{attribute 'linkalways'} 
{attribute 'no_explicit_call' := 'This FB is a CLASS and must be accessed using methods or properties'}
{attribute 'enable_dynamic_creation'}
FUNCTION_BLOCK GetBlueprintVisitor EXTENDS Disposable IMPLEMENTS I_NodePrototypeVisitor
VAR
	serializer : JsonSerializer;
END_VAR

METHOD VisitContent
VAR_INPUT
	VisitingContent : I_Content;
END_VAR
END_METHOD

METHOD VisitError
VAR_INPUT
	VisitingError : I_Alarm;
END_VAR
END_METHOD

METHOD VisitExtension
VAR_INPUT
	VisitingExtension : I_Extension;
END_VAR
END_METHOD

METHOD VisitInputPort
VAR_INPUT
	VisitingInputPort : I_InputPort;
END_VAR
END_METHOD

METHOD VisitMetadatum
VAR_INPUT
	VisitingMetadatum : I_Metadata;
END_VAR
END_METHOD

METHOD VisitNode
VAR_INPUT
	VisitingNode : I_Node;
END_VAR
serializer.StartObject();
END_METHOD

METHOD VisitOutputPort
VAR_INPUT
	VisitingOutputPort : I_OutputPort;
END_VAR
END_METHOD

METHOD VisitParameter
VAR_INPUT
	VisitingProperty : I_Parameter;
END_VAR
END_METHOD

METHOD VisitPrototype
VAR_INPUT
	VisitingPrototype : I_NodePrototype;
END_VAR
serializer.Reset();
serializer.StartObject();
serializer.AddKey('blueprints');
serializer.StartArray();

serializer.EndArray();
serializer.EndObject();
END_METHOD

END_FUNCTION_BLOCK

(* stored: Version 1.1.0.1, ProductVersion 3.1.4024.12
   POU GetBlueprintVisitor: Id {9f9a0116-9d81-4a08-a879-7a2851d51385}, SpecialFunc None
   Method VisitContent: Id {5d6b8e87-493f-4bc0-a416-bdda199c430d}
   Method VisitError: Id {08d6423b-3444-4d02-ae95-4e4c7fed218c}
   Method VisitExtension: Id {4b74c9d7-8e37-404e-add7-587af0696243}
   Method VisitInputPort: Id {0763b377-826e-4b34-9135-9701e00da90a}
   Method VisitMetadatum: Id {69ef5793-7e33-4a4a-bd31-0b8a852dd40c}
   Method VisitNode: Id {0c574603-4091-4b53-bc43-a99c409aff80}
   Method VisitOutputPort: Id {08afcd2c-2b3e-40a2-8371-470084bdd009}
   Method VisitParameter: Id {cb761164-ab6e-4c1f-a1c9-ed9d5f9c0450}
   Method VisitPrototype: Id {150c8dd2-723b-4895-862b-60480672d0cd} *)
